{attribute 'pack_mode' := '2'}
TYPE U_XTS_TRANSPORT_STATE :
UNION
  _st           : ST_XTS_TRANSPORT_STATE;
  _by   AT%I*   : ARRAY[1..SIZEOF(ST_XTS_TRANSPORT_STATE)] OF BYTE;
END_UNION
END_TYPE

(* stored: Version 1.1.0.1, ProductVersion 3.1.4024.12
   DUT U_XTS_TRANSPORT_STATE: Id {43029917-8e53-4a18-b5f1-2635668fe17e} *)
